{attribute 'qualified_only'}
TYPE E_Chamber1SingleProcessAbortPhase :
(
	StopAxes := 0,
	ResetAxes := 1
) UINT;
END_TYPE

(* stored: Version 1.1.0.1, ProductVersion 3.1.4026.18
   DUT E_Chamber1SingleProcessAbortPhase: Id {83d211fd-08e0-4362-9b31-1d7c9a3d1a95} *)
